FUNCTION_BLOCK ABSTRACT BaseParam EXTENDS Object IMPLEMENTS I_Param
VAR
	_display: STRING := '0';
END_VAR

//Base Param object.
// _display should be used to extract data from the interface in string form. 
// For example to use with visu.

//Q variable should be used to access the data directly from FB.
//Each derivative of this funciton should have added Q variable of literal type.

//Each derivative of BaseParam has Quick_Change(value) to directly modify Q value.

METHOD Change_Param
VAR_INPUT
	value	: STRING;
END_VAR
//How string value should be translated to other data type
END_METHOD

PROPERTY display : STRING
GET
display := _display;
END_GET
END_PROPERTY

END_FUNCTION_BLOCK

(* stored: Version 1.1.0.1, ProductVersion 3.1.4024.12
   POU BaseParam: Id {42da1c98-39da-4bba-9c49-2d1b281d511b}, SpecialFunc None
   Method Change_Param: Id {b2534efa-639f-4351-8c79-0b2100913693}
   Property display: Id {03aaf4e1-7807-4d0f-bfec-738b9c6ff2bb}
   Get Get: Id {53de3c53-9986-4265-90d7-e134a3cdb74f} *)
